ABB RobotStudio station: HandTracking_drawing.rspag

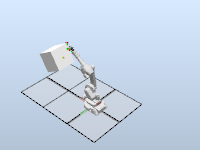
--- station ---
Station HandTracking (saved by RobotStudio 7.0.8743.626)
Controller Controller1
  mechanical unit ROB_1: IRB1600_6_145__02, 6 joints, base frame (0, 0, 0) mm
Layout (positions relative to the parent item):
  - IRB1600_6_145__02 [mechanism, from Robots\IRB1600_6_145_G_02.rslib] at (0, 0, 0) mm; joint values [0, 0.0197, -0.6431, -3.1416, 0.0172, 3.1416] (rad or m)
  - Part_1 [part] at (201, 0, 301) mm
  - Pen [mechanism, from Training Objects\Pen.rslib] at (703.05, 0, 1575.48) mm, rotated rx 0 ry 53.3 rz 0 deg
Attachment: Pen is attached to IRB1600_6_145__02 / Link6
Targets, tools, work objects and paths stored in the station and not in the controller backup, written as RAPID:
! task T_ROB1
MODULE Module1
  PROC Path_10()
    MoveJ home,v1000,z100,Pen_TCP\WObj:=wobj0;
  ENDPROC
ENDMODULE


--- Backups/Controller1/RAPID/TASK1/PROGMOD/CalibData.mod ---
MODULE CalibData
	PERS tooldata Pen_TCP:=[TRUE,[[110,0,140],[0.707106781,0,0.707106781,0]],[1,[10.7435139,0,140],[1,0,0,0],0,0,0]];
ENDMODULE

--- Backups/Controller1/RAPID/TASK1/PROGMOD/Module1.mod ---
MODULE Module1
	CONST robtarget home:=[[881.040805141,0,1570.963328368],[0.31485624,0,0.949139372,0],[0,-1,-1,1],[9E+09,9E+09,9E+09,9E+09,9E+09,9E+09]];
    CONST robtarget Target_20:=[[300,300,0],[0.707106781,0,0,0.707106781],[1,0,0,0],[9E+09,9E+09,9E+09,9E+09,9E+09,9E+09]];
    PERS num bReachable:=1;
    TASK PERS wobjdata myframe:=[FALSE,TRUE,"",[[1300,-300,1419.615],[0.353553391,-0.612372436,0.612372436,-0.353553391]],[[0,0,0],[1,0,0,0]]];
    VAR num operatingmode:=0;
    VAR num waitpaint:=0;

    !Made by Luka Dragar
    !Follow me @thelukadragar
    !
    !Thanks to ABB forum
    !
    !
    !
    !




    PROC main()
        VAR socketdev server_socket;
        VAR socketdev client_socket;
        VAR string receive_string;
        VAR string receive_string2;
        VAR string client_ip;
        VAR robtarget mytr;
        VAR string myIP:= "127.0.0.1"; !same as in config.py !!!



        SocketCreate server_socket;
        SocketBind server_socket,myIP, 55555;
        SocketListen server_socket;

        ConfL\Off;
        ConfJ\Off;

        MoveJ home,v1000,z30,Pen_TCP\WObj:=wobj0;


        ! Waiting for a connection request
         SocketAccept server_socket, client_socket\ClientAddress:=client_ip\Time:=WAIT_MAX;
         SocketSend client_socket \Str :="Robot at position "+TargetToString(home);

        WHILE TRUE DO
            !waiting to recive
            SocketReceive client_socket \Str := receive_string2;

            IF receive_string2="xy" THEN
                !operating mode is in xy plane
                operatingmode:=0;
                SocketSend client_socket \Str :="Robot set to move in XY plane";
                waitpaint:=1;

                TPWrite"moving set to XY plane now";

            ELSEIF receive_string2="xyz" THEN
                !operating mode is in xyz plane
                operatingmode:=1;
                waitpaint:=0;
                SocketSend client_socket \Str :="Robot set to move in XYZ !";
                TPWrite"moving set to XYZ now !";
                Reset doPaint;

            ELSE
                !MOVE



                IF waitpaint<3 AND operatingmode=0 THEN
                    waitpaint:=waitpaint+1;
                ELSE
                    IF waitpaint=3 THEN
                    Set doPaint;
                    waitpaint:=0;
                 ENDIF

                ENDIF

                 mytr:= StringToTargetFromxy(receive_string2); !get target from string
                 move mytr;!check if is reachable then move
            ENDIF
        ENDWHILE


    ERROR
        IF ERRNO=ERR_SOCK_TIMEOUT THEN
            RETRY;

        ELSEIF ERRNO=ERR_SOCK_CLOSED THEN

        SocketCreate server_socket;
        SocketBind server_socket, myIP, 55555;
        SocketListen server_socket;
            RETRY;
        ELSE
            RETRY;

        ENDIF
    UNDO
        SocketClose server_socket;
        SocketClose client_socket;
    ENDPROC


     FUNC robtarget create_robtarget(pos position)
       RETURN [position,[0.707106781,0,0,0.707106781],[1,0,0,0],[9E9,9E9,9E9,9E9,9E9,9E9]];
    ENDFUNC

    FUNC string TargetToString(robtarget target)
    VAR string tmpString;
    !pos data
    tmpString:=NumToStr (target.trans.x,0);
    AddToString tmpString,target.trans.y;
    AddToString tmpString, target.trans.z;
    ! orient data
    AddToString tmpString, target.rot.q1;
    AddToString tmpString, target.rot.q2;
    AddToString tmpString, target.rot.q3;
    AddToString tmpString, target.rot.q4;
    ! conf data
    AddToString tmpString, target.robconf.cf1;
    AddToString tmpString, target.robconf.cf4;
    AddToString tmpString, target.robconf.cf6;
    AddToString tmpString, target.robconf.cfx;
RETURN tmpString;
ENDFUNC

FUNC robtarget StringToTarget(string value)
    !CAN BE USED IF OREANTATIONS ARE NEEDED CURENTLY NOT USED
VAR robtarget tmpTarget;
VAR bool bResult;
VAR num posX;
VAR num posY;
VAR num posZ;
VAR num posQ1;
VAR num posQ2;
VAR num posQ3;
VAR num posQ4;
VAR num poscf1;
VAR num poscf4;
VAR num poscf6;
VAR num poscfx;
! Find split positions in string

posX:=StrFind (value, 1,";");
posY:=StrFind (value, posX+1,";");
posZ:=StrFind (value, posY+1,";");
posQ1:=StrFind (value, posZ+1,";");
posQ2:=StrFind(value, posQ1+1,";");
posQ3:=StrFind (value,posQ2+1,";");
posQ4:=Strfind(value, posQ3+1,";");
poscf1:=StrFind(value, posQ4+1,";");
poscf4:=StrFind(value, poscf1+1,";");
poscf6:=StrFind(value, poscf4+1,";");
poscfx:=StrFind(value,poscf6+1, ";");
! read all strings
! pos data
bResult:=StrToval(StrPart(value,1,posX-1), tmpTarget.trans.x);
bResult:=StrToVal(StrPart(value,posX+1, posY-posX-1), tmpTarget.trans.y);
bResult:=StrToVal(StrPart(value,posY+1, posZ-posY -1), tmpTarget.trans.z);
! orient data
bResult:=StrToVal(StrPart(value, posZ+1, posQ1-posz-1), tmpTarget.rot.q1);
bResult:=StrToval (StrPart(value,posQ1+1, posQ2-posQ1-1), tmpTarget.rot.q2);
bResult:=StrToVal(StrPart(value,posQ2+1, posQ3-posQ2-1), tmpTarget.rot.q3);
bResult:=StrToVal(StrPart(value,posQ3+1,posQ4-posQ3-1), tmpTarget.rot.q4);
! conf data
bResult:=StrToVal(StrPart(value,posQ4+1, poscf1-posQ4-1), tmpTarget.robconf.cf1);
bResult:=StrToVal(StrPart(value, poscf1+1,poscf4-poscf1-1), tmpTarget.robconf.cf4);
bResult:=StrToval(StrPart(value,poscf4+1,poscf6-poscf4-1), tmpTarget.robconf.cf6);
bResult:=StrToVal(StrPart(value,poscf6+1,poscfx-poscf6-1), tmpTarget.robconf.cfx);
RETURN tmpTarget;

ERROR
    RETURN Target_20;



ENDFUNC

FUNC robtarget StringToTargetFromxy(string value)
VAR pos tmpPos;
VAR robtarget tmpTarget;
VAR bool bResult;
VAR num posX;
VAR num posY;
VAR num posZ;
VAR num posQ1;
VAR num posQ2;
VAR num posQ3;
VAR num posQ4;
VAR num poscf1;
VAR num poscf4;
VAR num poscf6;
VAR num poscfx;
VAR num xxx;
VAR num yyy;
VAR num zzz:=0;
! Find split positions in string

posX:=StrFind (value, 1,";");
posY:=StrFind (value, posX+1,";");
IF operatingmode=1 THEN
posZ:=StrFind (value, posY+1,";");
ENDIF

! pos data
bResult:=StrToval(StrPart(value,1,posX-1), tmpPos.x);
tmpPos.x:=-tmpPos.x;
bResult:=StrToVal(StrPart(value,posX+1, posY-posX-1), tmpPos.y);

IF operatingmode=1 THEN
bResult:=StrToVal(StrPart(value,posY+1, posZ-posY -1), tmpPos.z);
ELSE
tmpPos.z:=zzz; !z is set to 0
ENDIF
tmpTarget:=create_robtarget(tmpPos);
RETURN tmpTarget;

ERROR
    RETURN Target_20;!middle target of error
ENDFUNC

PROC AddToString(INOUT string inString,num value)
inString:=inString+";"+NumToStr(value,0);
ENDPROC

PROC move(robtarget target)
    CheckReachable target,Pen_TCP;
           IF bReachable=2 THEN
                !notreachable
                TPWrite"not reachable";
           ELSEIF bReachable=1 THEN
                !reachable start moving
                MoveJ target,v2000,z10,Pen_TCP\WObj:=myframe;
          ENDIF
    ERROR
        TPWrite"error in move";

ENDPROC


 PROC CheckReachable(robtarget myRobtarget,PERS tooldata ToolReach1,\PERS wobjdata WobjReach1)

      VAR jointtarget jntReach1;
      bReachable:=1;
      IF Present(WobjReach1) THEN
            jntReach1:=CalcJointT(myRobtarget,ToolReach1\WObj:=WobjReach1);
      ELSE
            jntReach1:=CalcJointT(myRobtarget,ToolReach1);
      ENDIF
      RETURN;
      ERROR
         IF ERRNO=ERR_OUTSIDE_REACH THEN
                bReachable:=2;
               TRYNEXT;
        ENDIF
         IF ERRNO=ERR_ROBLIMIT THEN
                bReachable:=2;
               TRYNEXT;
        ENDIF
        bReachable:=2;
        RETURN;
  ENDPROC
ENDMODULE

--- Backups/Controller1/SYSPAR/EIO.cfg ---
EIO:CFG_1.0:6:1::
#
EIO_SIGNAL:

      -Name "doPaint" -SignalType "DO" -Label "paint"
